{attribute 'qualified_only'}
{attribute 'strict'}
TYPE E_MACHINE_POSITIONS :
(
	eHome := 0,
	ePosition1 := 1,
	ePosition2 := 2,
	ePosition3 := 3,
	ePosition4 := 4
);
END_TYPE

(* stored: Version 1.1.0.1, ProductVersion 3.1.4024.3
   DUT E_MACHINE_POSITIONS: Id {b2def280-f0b1-487d-9f8c-be4f3562f0bc} *)
